// TIA Portal V19 export
TYPE "C701_VAR_IF_KMI_TYPIC"
   STRUCT
      EXT_AUT { ExternalAccessible := 'False'; ExternalVisible := 'False'; ExternalWritable := 'False'} : Bool;   // Externe (hoofd) beveiliging aangesproken
      EXT_HW { ExternalAccessible := 'False'; ExternalVisible := 'False'; ExternalWritable := 'False'} : Bool;   // Sturings hardware (PLC) in storing
      STO { ExternalAccessible := 'False'; ExternalVisible := 'False'; ExternalWritable := 'False'} : Struct   // Opsomming van alle storingen en meldingen
         A001 : Bool;   // Storing algemeen luchtbehandelingssysteem
         A002 : Bool;   // Storing algemeen koelmachine
         A003 : Bool;   // Storing algemeen warmtepomp
         A004 : Bool;   // Storing brandklep gesloten
         A005 : Bool;   // Storing temperatuur besturingslokaal
         A006 : Bool;   // Storing algemeen besturingslokaal
         A007 : Bool;   // Storing temperatuur opleidings/trainer/test/pauze lokaal
         A008 : Bool;   // Storing algemeen opleidings/trainer/test/pauze lokaal
         A009 : Bool;   // Storing temperatuur vergaderzaal/kantoor
         A010 : Bool;   // Storing algemeen vergaderzaal/kantoor
         A011 : Bool;   // Storing temperatuur batterijlokaal
         A012 : Bool;   // Storing algemeen batterijlokaal
         A013 : Bool;   // Storing temperatuur astrid/gsm lokaal
         A014 : Bool;   // Storing algemeen astrid/gsm lokaal
         A015 : Bool;   // Storing temperatuur sanitaire ruimte
         A016 : Bool;   // Storing algemeen sanitaire ruimte
         AT01 : Bool;
         AT02 : Bool;
         M001 : Bool;
         M002 : Bool;
      END_STRUCT;
   END_STRUCT;
END_TYPE
